FUNCTION_BLOCK SmartMotor 

VAR
	errorID: INT ;
    isError: BOOL ;
    isReady : BOOL;
	
	isReset : BOOL := FALSE;
END_VAR


    errorID:= 6589 ;
    isError:= TRUE ;
    isReady := FALSE;


 IF isReset THEN
	 ActReset();
 END_IF

ACTION ActReset:
// Action: Act_Reset (Under FB_SmartMotor)
	errorID:= 0;
    isError:= FALSE ;
    isReady := TRUE;
END_ACTION

END_FUNCTION_BLOCK

(* stored: Version 1.1.0.1, ProductVersion 3.1.4024.16
   POU SmartMotor: Id {87310dc6-ef4d-44c3-a7ed-d147a629e919}, SpecialFunc None
   Action ActReset: Id {5bc79f0a-a8d1-484d-b22f-10f825f9de79} *)
